// TIA Portal V20 export
TYPE "LKinCtrl_typeCOffOutNextButOneCmd"
   STRUCT
      transitionParameter : Array[1..5] of LReal;   // blending parameters
   END_STRUCT;
END_TYPE
